ABB RobotStudio station: HCV_1_20220901-201702.rsstn

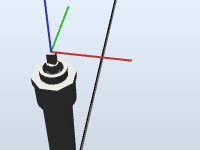
Station HCV (saved by RobotStudio 6.5.7558.2005)
Layout (positions relative to the parent item):
  - HCV [mechanism, from Libraries\HCV.rslib] at (0, 0, 0) mm
